TYPE MEMBERSHIP_FUNCTION :
	STRUCT
		Name:STRING;
		Shape: MF_SHAPE;//membership function shape
		//MfPoints: ARRAY[*]OF REAL;//membership funciton points
		Points: ARRAY[1..5]OF REAL;
	END_STRUCT
END_TYPE

(* stored: Version 1.1.0.1, ProductVersion 3.1.4024.6
   DUT MEMBERSHIP_FUNCTION: Id {20a606ee-cf60-4797-a527-0a6c9c518a98} *)
